TEXTLIST WorkAreaState
  0 = 'F+D'
  1 = 'O+D'
  2 = 'F+Wg'
  3 = 'O+Wg'
  4 = 'O+Wd'
  5 = 'O+Wd+D'
  6 = 'O+Tg'
  7 = 'O+Tg+D'
  8 = 'O+Td'
  9 = 'O+Td+D'
  10 = 'O+E'
  11 = 'O+E+D'
  12 = 'O+Lr'
  13 = 'O+Lr+D'
  14 = 'O+Li'
  15 = 'O+Li+D'
  16 = 'O+Le'
  17 = 'O+Le+D'
   = ''
END_TEXTLIST

(* stored: Version 1.1.0.1, ProductVersion 3.1.4024.11
   TextList WorkAreaState: Id {66844c70-6742-42e4-accd-833470415824} *)
